(* CODESYS project projects

Project tree, tasks and I/O mapping:
  Device : CODESYS Control for Raspberry Pi SL, CODESYS GmbH, order no. 2302000009, version 4.7.0.0
    application Application
      libraries: Standard, 3.5.18.0 (System); CmpBitmapPool, * (System)
      task AC_RMP_Task (cyclic, interval t#20ms, priority 30) calls AC_PRG_RMP
      task EtherCAT_Task (cyclic, interval t#4ms, priority 1) calls nothing
      task HIGH (cyclic, interval t#5ms, priority 1) calls AC_CALL_HIGH_START, AC_CALL_HIGH_END
      task LOW (cyclic, interval t#20ms, priority 10) calls AC_CALL_LOW_START, AC_CALL_LOW_END
      task MainTask (cyclic, interval t#4ms, priority 1) calls Climate, Environment
      task TrendRecordingTask (cyclic, interval 100 ms, priority 31) calls VisuTrendStorageAccess.GlobalInstances.g_TrendRecordingManager.CyclicCall
      task VISU_TASK (cyclic, interval 100 ms, priority 31) calls VisuElems.Visu_Prg
      AC_FBs/
        function block AC_PersistenceManager [ST]
        function block AC_PersistenceManager_PersistenceChannel [ST]
      AC_RMP/
        program AC_PRG_RMP [ST]
        global variables AC_RMP
      AC_Std/
        program AC_CALL_HIGH_END [ST]
        program AC_CALL_HIGH_START [ST]
        program AC_CALL_LOW_END [ST]
        program AC_CALL_LOW_START [ST]
        function AC_Init [ST]
        function AC_InitInternal [ST]
        function AC_OnlineChange [ST]
        global variables GVL_MODULE_TREE
        global variables GVL_PersistenceManager
        global variables MODULE_INFOS
      program Climate [CFC]
      Enumerated Types/
        data type etAlarmTypes
      program Environment [CFC]
      Function Blocks/
        function block FB_Meter [ST]: rCalcAverage, rCalcMaximum, rCalcMinimum, rScaleOutput, xAlarms, xReset
      Images/
        image pool ImagePool
      Interfaces/
        interface itfMeter: rCalcAverage, rCalcMaximum, rCalcMinimum, rScaleOutput, xAlarms, xReset
      program Irrigation [CFC]
      program Lighting [CFC]
      text PersistenceConfig
      visualisation SimpleMeter
      Structured Types/
        data type stAlarm
      Trend Recording Manager
        Visualization_Trend1
      visualisation vbMeter
      program Ventilation [CFC]
      visualisation Visualization
    Camera device
      <Empty>
    EtherCAT_Master : EtherCAT Master, 3S - Smart Software Solutions GmbH, version 4.5.0.0
        settings: NetworkName = 'eth0'; NetworkName = "eth0"; SrcAddress1 = 56486; SrcAddress2 = 850751358
      EK1100 : EK1100 EtherCAT Coupler (2A E-Bus), Beckhoff Automation GmbH & Co. KG, order no. EK1100, version Revision=16#00120000
          settings: StationAlias = 0; DC sync0 cycletime = 4000; DC sync1 cycletime = 4000
        EL1018 : EL1018 8Ch. Dig. Input 24V, 10µs, Beckhoff Automation GmbH & Co. KG, order no. EL1018, version Revision=16#00120000
            settings: StationAlias = 0; DC sync0 cycletime = 4000; DC sync1 cycletime = 4000
            unmapped channels: Input, Input, Input, Input, Input, Input, Input, Input
        EL2008 : EL2008 8Ch. Dig. Output 24V, 0.5A, Beckhoff Automation GmbH & Co. KG, order no. EL2008, version Revision=16#00100000
            settings: StationAlias = 0; DC sync0 cycletime = 4000; DC sync1 cycletime = 4000
            unmapped channels: Output, Output, Output, Output, Output, Output, Output, Output
        EL3152 : EL3152 2Ch. Ana. Input 4-20mA, Beckhoff Automation GmbH & Co. KG, order no. EL3152, version Revision=16#00000000
            settings: StationAlias = 0; DC sync0 cycletime = 4000; DC sync1 cycletime = 4000
            input  Transmitter101 : INT  // Value
            unmapped channels: Status, Status, Value
    GPIOs_A_B : GPIOs A/B, 3S - Smart Software Solutions GmbH, version 4.7.0.0
        unmapped channels: digital inputs (GPIO0..GPIO31), digital outputs (GPIO0..GPIO31)
    I²C
    Onewire
      Onewire_master : Onewire master, 3S - Smart Software Solutions GmbH, version 4.7.0.0
        AmbTemp101 : DS18B20, 3S - Smart Software Solutions GmbH, version 4.7.0.0
            settings: Unique device address = '28-3ce1045748ac'
        SoilTemp101 : DS18B20, 3S - Smart Software Solutions GmbH, version 4.7.0.0
            settings: Unique device address = '28-3ce1045771af'
        SoilTemp102 : DS18B20, 3S - Smart Software Solutions GmbH, version 4.7.0.0
            settings: Unique device address = '28-3ce10457587b'
        SoilTemp103 : DS18B20, 3S - Smart Software Solutions GmbH, version 4.7.0.0
            settings: Unique device address = '28-3ce104579414'
    SoftMotion General Axis Pool
    SPI
  libraries: VisuSymbols, 4.4.0.0 (System); AC_Persistence, 4.2.0.0 (3S - Smart Software Solutions GmbH)
  5ce3da45-db07-42e7-a21c-a00fff4ed8f6|Humidity.svg
  5ce3da45-db07-42e7-a21c-a00fff4ed8f6|Humidity.svg
  5ce3da45-db07-42e7-a21c-a00fff4ed8f6|Moisture.svg
  5ce3da45-db07-42e7-a21c-a00fff4ed8f6|Moisture.svg
  5ce3da45-db07-42e7-a21c-a00fff4ed8f6|Succulents.jpg
  5ce3da45-db07-42e7-a21c-a00fff4ed8f6|Succulents.jpg
  5ce3da45-db07-42e7-a21c-a00fff4ed8f6|Thermometer.svg
  5ce3da45-db07-42e7-a21c-a00fff4ed8f6|Thermometer.svg
  AC_GENERATOR_DATA
  text list GlobalTextList
  PersistenceManager
    Channels (pChannels)
      PersistenceChannel
        ASCIIFileStorage
        Data Storage (itfDataStorage)
  text list System
*)

// Device/Application/Enumerated Types/etAlarmTypes
{attribute 'qualified_only'}
{attribute 'strict'}
TYPE etAlarmTypes :
(
	UR := 0, // Under range alarm
	LL := 1, // Low low alarm
	L := 2, // Low Alarm
	H := 3, // High Alarm
	HH := 4, // High High Alarm
	OVR := 5 // Overage Range Alarm
);
END_TYPE

// Device/Application/Structured Types/stAlarm
TYPE stAlarm :
STRUCT
	
END_STRUCT
END_TYPE

// Device/Application/AC_RMP/AC_RMP
//Code generated by Application Composer.
//Modifying generated code is not recommended!
{attribute 'global_init_slot' := '60000'}
{attribute 'init_on_onlchange'}

VAR_GLOBAL
	{attribute 'init_on_onlchange'}
	AC_RMP_Service: AC_PERSIST.AC.RMPService := (uiLocalAppID:=9744, uiNumberOfConnections:=0, pSendConnection:=0, pReceiveConnection:=0, pRMPComFB:=0);
END_VAR

// Device/Application/AC_Std/GVL_MODULE_TREE
//Code generated by Application Composer.
//Modifying generated code is not recommended!

VAR_GLOBAL
	Module_Tree: AC_PERSIST.AC.ModuleTree;
	aNodes: ARRAY[0..3] OF AC_PERSIST.AC.MNode;
	AC_Environment: AC_PERSIST.AC.MEnv;
END_VAR

// Device/Application/AC_Std/GVL_PersistenceManager
//Code generated by Application Composer.
//Modifying generated code is not recommended!
{attribute 'analysis' := '-103'}

VAR_GLOBAL
	PersistenceManager: AC_PersistenceManager;
END_VAR

// Device/Application/AC_Std/MODULE_INFOS
//Code generated by Application Composer.
//Modifying generated code is not recommended!
{attribute 'global_init_slot' := '40000'}
{attribute 'init_on_onlchange'}

VAR_GLOBAL
	{attribute 'init_on_onlchange'}
	AC_PERSIST_PersistenceManager_INFO: AC_PERSIST.AC.ModuleInfo := (pbyModuleType := ADR('AC_PERSIST.PersistenceManager'));
	{attribute 'init_on_onlchange'}
	AC_PERSIST_PersistenceChannel_INFO: AC_PERSIST.AC.ModuleInfo := (pbyModuleType := ADR('AC_PERSIST.PersistenceChannel'));
	{attribute 'init_on_onlchange'}
	AC_PERSIST_ASCIIFileStorage_INFO: AC_PERSIST.AC.ModuleInfo := (pbyModuleType := ADR('AC_PERSIST.ASCIIFileStorage'));
END_VAR

// Device/Application/AC_RMP/AC_PRG_RMP
//Code generated by Application Composer.
//Modifying generated code is not recommended!
{attribute 'analysis' := '-9'}
PROGRAM AC_PRG_RMP
VAR
    itfRmpService2 : AC_PERSIST.AC.IRmpService2 := 0;
    xStartCyclicAction : BOOL;
    xIsActionOngoing : BOOL;
    xValid : BOOL;
    xValidEnd : BOOL := TRUE;
END_VAR

//Code generated by Application Composer.
//Modifying generated code is not recommended!
__QUERYINTERFACE(AC_RMP_Service, itfRmpService2);
IF itfRmpService2 <> 0 AND xValidEnd THEN
    xValid := itfRmpService2.GetIsActionOngoing(xIsActionOngoing=>xIsActionOngoing);
    IF NOT xValid OR (xValid AND xIsActionOngoing) THEN
        xStartCyclicAction := FALSE;
    ELSE
        xStartCyclicAction := itfRmpService2.SetIsActionOngoing(TRUE);
    END_IF
ELSE
    xStartCyclicAction := TRUE;
END_IF
IF xStartCyclicAction THEN
    AC_RMP_Service.CyclicCall() ;
END_IF
IF itfRmpService2 <> 0 AND (xStartCyclicAction OR NOT xValidEnd) THEN
    xValidEnd := itfRmpService2.SetIsActionOngoing(FALSE);
END_IF

END_PROGRAM

// Device/Application/AC_Std/AC_CALL_HIGH_START
//Code generated by Application Composer.
//Modifying generated code is not recommended!
{attribute 'analysis' := '-6, -9'}
PROGRAM AC_CALL_HIGH_START

//Code generated by Application Composer.
//Modifying generated code is not recommended!
PersistenceManager.CallPrioHighStart() ;

END_PROGRAM

// Device/Application/AC_Std/AC_CALL_HIGH_END
//Code generated by Application Composer.
//Modifying generated code is not recommended!
{attribute 'analysis' := '-6, -9'}
PROGRAM AC_CALL_HIGH_END

//Code generated by Application Composer.
//Modifying generated code is not recommended!
PersistenceManager.CallPrioHighEnd() ;

END_PROGRAM

// Device/Application/AC_Std/AC_CALL_LOW_START
//Code generated by Application Composer.
//Modifying generated code is not recommended!
{attribute 'analysis' := '-6, -9'}
PROGRAM AC_CALL_LOW_START

//Code generated by Application Composer.
//Modifying generated code is not recommended!
PersistenceManager.CallPrioLowStart() ;

END_PROGRAM

// Device/Application/AC_Std/AC_CALL_LOW_END
//Code generated by Application Composer.
//Modifying generated code is not recommended!
{attribute 'analysis' := '-6, -9'}
PROGRAM AC_CALL_LOW_END

//Code generated by Application Composer.
//Modifying generated code is not recommended!
PersistenceManager.CallPrioLowEnd() ;

END_PROGRAM

// Device/Application/Climate
PROGRAM Climate
VAR
	rAmbTempSensor : ARRAY[101..103] OF fb_meter; // Ambient temperature probes
	iAmbRosemountSensor : INT; 
END_VAR

// parameter rAmbTempSensor[102].iInterval := T#5s
// parameter rAmbTempSensor[102].rOut_100 := 257
// parameter rAmbTempSensor[102].rOut_0 := -67
// parameter rAmbTempSensor[102].rIn_100 := 125
// parameter rAmbTempSensor[102].rIn_0 := -55
// parameter rAmbTempSensor[102].sDateLastServiced := ''
// parameter rAmbTempSensor[102].sSerial := ''
// parameter rAmbTempSensor[102].sUnits := ''
// parameter rAmbTempSensor[102].sDescription := ''
// parameter rAmbTempSensor[102].sName := ''
// parameter rAmbTempSensor[102].rHHLimit := 95
// parameter rAmbTempSensor[102].rHLimit := 90
// parameter rAmbTempSensor[102].rLLimit := 48
// parameter rAmbTempSensor[102].rLLLimit := 32
// parameter rAmbTempSensor[102].rURLimit := -5
// parameter rAmbTempSensor[102].tOVRAlarm := T#5s
// parameter rAmbTempSensor[102].tHHAlarm := T#5s
// parameter rAmbTempSensor[102].tHAlarm := T#5s
// parameter rAmbTempSensor[102].tLAlarm := T#5s
// parameter rAmbTempSensor[102].tLLAlarm := T#5s
// parameter rAmbTempSensor[102].tURAlarm := T#5s
rAmbTempSensor[102](xEnable := true, rIn := Transmitter101); // FB_METER
// parameter rAmbTempSensor[101].iInterval := T#5s
// parameter rAmbTempSensor[101].rOut_100 := 257
// parameter rAmbTempSensor[101].rOut_0 := -67
// parameter rAmbTempSensor[101].rIn_100 := 125
// parameter rAmbTempSensor[101].rIn_0 := -55
// parameter rAmbTempSensor[101].sDateLastServiced := ''
// parameter rAmbTempSensor[101].sSerial := ''
// parameter rAmbTempSensor[101].sUnits := ''
// parameter rAmbTempSensor[101].sDescription := ''
// parameter rAmbTempSensor[101].sName := ''
// parameter rAmbTempSensor[101].rHHLimit := 95
// parameter rAmbTempSensor[101].rHLimit := 90
// parameter rAmbTempSensor[101].rLLimit := 48
// parameter rAmbTempSensor[101].rLLLimit := 32
// parameter rAmbTempSensor[101].rURLimit := -5
// parameter rAmbTempSensor[101].tOVRAlarm := T#5s
// parameter rAmbTempSensor[101].tHHAlarm := T#5s
// parameter rAmbTempSensor[101].tHAlarm := T#5s
// parameter rAmbTempSensor[101].tLAlarm := T#5s
// parameter rAmbTempSensor[101].tLLAlarm := T#5s
// parameter rAmbTempSensor[101].tURAlarm := T#5s
rAmbTempSensor[101](xEnable := true, rIn := AmbTemp101.rTemp); // FB_METER

END_PROGRAM

// Device/Application/Function Blocks/FB_Meter
FUNCTION_BLOCK FB_Meter IMPLEMENTS itfMeter
VAR_INPUT
	xEnable : BOOL; 
	rIn : LREAL; 
	xResetCalcs : BOOL; 
END_VAR
VAR_OUTPUT
	rOut, rMin, rMax, rAvg : REAL; 
	xInAlarm, xBusy, xDone, xError : BOOL; 
	sStatus : STRING; // Status of function block
END_VAR
VAR
	tonUr, tonLL, tonL, tonH, tonHH, tonOVR : TON; 
	{attribute 'ac_persist' := 'PersistenceChannel'}
	xURActive, xLLActive, xLActive, xHActive, xHHActive, xOVRActive : BOOL; 
	rIn_PCT : REAL; // REAL INPUT EXPRESSED AS PERCENTAGE
	i : INT; 
	{attribute 'ac_persist' := 'PersistenceChannel'}
	iExecutions : DINT; 
	iMod : INT; 
END_VAR
VAR_INPUT CONSTANT
	{attribute 'parameterCategory':='Alarming'}
	tURAlarm,tLLAlarm,tLAlarm,tHAlarm,tHHAlarm,tOVRAlarm : TIME := T#5S; // Alarm Time duration
	{attribute 'ac_persist' := 'PersistenceChannel'}
	{attribute 'parameterCategory':='Alarming'}
	rURLimit : REAL := -5.0; 
    {attribute 'ac_persist' := 'PersistenceChannel'}
	{attribute 'parameterCategory':='Alarming'}
	rLLLimit : REAL := 32.0; 
	{attribute 'ac_persist' := 'PersistenceChannel'}
	{attribute 'parameterCategory':='Alarming'}
	rLLimit  : REAL := 48.0; 
	{attribute 'ac_persist' := 'PersistenceChannel'}
	{attribute 'parameterCategory':='Alarming'}
	rHLimit  : REAL := 90.0; 
	{attribute 'ac_persist' := 'PersistenceChannel'}
    {attribute 'parameterCategory':='Alarming'}
	rHHLimit : REAL := 95.0; 
	{attribute 'ac_persist' := 'PersistenceChannel'}
	{attribute 'parameterCategory':='Alarming'}
	rOVRLimit : REAL := 125; // Alarm limits
	{attribute 'ac_persist' := 'PersistenceChannel'}
	{attribute 'parameterCategory':='Alarming'}
	xarEnableAlarms: ARRAY [0..5] OF BOOL := [2(FALSE), 2(TRUE), 2(FALSE)];
	{attribute 'ac_persist' := 'PersistenceChannel'}
	{attribute 'parameterCategory':='Information'}
	sName, sDescription, sUnits, sSerial, sDateLastServiced : STRING; 
	{attribute 'ac_persist' := 'PersistenceChannel'}
	{attribute 'parameterCategory':='Scaling'}
	rIn_0 : REAL := 4; // VALUE AT 0 PERCENT INPUT
	{attribute 'ac_persist' := 'PersistenceChannel'}
	{attribute 'parameterCategory':='Scaling'}
	rIn_100 : REAL := 20; // VALUE AT 100 PERCENT INPUT
	{attribute 'ac_persist' := 'PersistenceChannel'}
	{attribute 'parameterCategory':='Scaling'}
	rOut_0 : REAL := 0; // Output at 0 percent
	{attribute 'ac_persist' := 'PersistenceChannel'}
	{attribute 'parameterCategory':='Scaling'}
	rOut_100 : REAL := 100;  // Output at 100 percent
	{attribute 'ac_persist' := 'PersistenceChannel'}
	{attribute 'parameterCategory':='Time'}
	iInterval : TIME := t#5s; 
END_VAR

// Run the calculations
// iMod := (to_int(time()) MOD TO_INT(iInterval)); 
IF TRUE (*(TO_INT(TIME()) MOD TO_INT(iInterval)) = 0*) THEN
	iExecutions := iExecutions+1; 
	rCalcAverage(rIn:=rOut,iExecutions:=iExecutions); 
	rCalcMaximum(rIn:=rOut); 
	rCalcMinimum(rin:=rOut); 
	rScaleOutput(rIn:=rIn); 
// From the list of enabled alarms, calculate the alarm expression
	FOR i:=0 TO 5 DO
		IF i<=2 THEN 
			xAlarms(rIn:=rIn,iAlarmType:=etAlarmTypes.L); 
		ELSIF i>=3 AND i<6 THEN 
			xAlarms(rIN:=rIn,iAlarmType:=etAlarmTypes.H); 
		ELSE
			; 
		END_IF	
	END_FOR
END_IF
	
IF xResetCalcs THEN 
	xReset(); 
END_IF

{warning 'Add method implementation '}
METHOD rCalcAverage : REAL
VAR_INPUT
	rIn	: REAL;
	iExecutions : DINT; 
END_VAR
VAR_OUTPUT
END_VAR
rAvg:=(rAvg*iExecutions+MAX(RAvg,rIn))/(iExecutions+1); // calculate the average of the output
END_METHOD

{warning 'Add method implementation '}
METHOD rCalcMaximum : REAL
VAR_INPUT
	rIn	: REAL;
END_VAR
IF rIn > rMax THEN 
	rMax := rIN;
ELSE 
	rMax := rMax; 
END_IF
END_METHOD

{warning 'Add method implementation '}
METHOD rCalcMinimum : REAL
VAR_INPUT
	rIn	: REAL;
END_VAR
IF rIn < rMin THEN 
	rMin := rIn; 
ELSE
	rMin := rMin; 
END_IF
END_METHOD

{warning 'Add method implementation '}
METHOD rScaleOutput : REAL
VAR_INPUT
	rIn	: REAL;
END_VAR
THIS^.rIn_PCT:=(rIn-rIn_0)/(rIn_100-rIn_0)*100; // Calculate output in percentage
this^.rOut:=THIS^.rIn_PCT/100 * (THIS^.rOut_100 - THIS^.rOut_0) + THIS^.rOut_0; // Linear scaling of output within scaling parameters
END_METHOD

{warning 'Add method implementation '}
METHOD xAlarms : BOOL
VAR_INPUT
	rIn	: REAL;
	(* Alarm Type *)
	iAlarmType	: etAlarmTypes;
END_VAR
IF iAlarmType = etAlarmTypes.L THEN 
	IF rIn <= rURLimit THEN 
		xURActive := TRUE; 
		tonUR(in:=TRUE,PT:=tURAlarm); 
	ELSIF rIn<=rLLLimit THEN 
		xLLActive := TRUE; 
		tonLL(in:=TRUE,PT:=tLLAlarm); 
	ELSIF rIn<=rLLimit THEN 
		xLActive := TRUE; 
		tonL(in:=TRUE,pt:=TLAlarm); 
	ELSE
		xURActive:=xLLActive:=xLActive:=FALSE;
		tonUR(in:=FALSE); 
	 	tonLL(in:=FALSE); 
		tonL(in:=FALSE); 
	END_IF
ELSIF iAlarmType = etAlarmTypes.H THEN 
	IF rIn >= rHLimit THEN 
		xHActive := TRUE; 
		tonH(in:=TRUE,pt:=tHAlarm); 
	ELSIF rIn >= rHHLimit THEN 
		xHHActive := TRUE; 
		tonHH(in:=TRUE,PT:=tHHAlarm); 
	ELSIF rIn >= rOVRLimit THEN 
		xOvrActive := TRUE; 
		tonOvr(in:=TRUE,PT:=tOvrAlarm); 
	ELSE
		xHActive:=xHHActive:=xOVRActive:=FALSE; 
		tonH(in:=FALSE); 
		tonHH(in:=FALSE); 
		tonOVR(in:=FALSE); 
	END_IF
END_IF
END_METHOD

{warning 'Add method implementation '}
METHOD xReset : BOOL
THIS^.iExecutions:=0; 
rOut:=rMin:=rMax:=rAvg:=0; 
xResetCalcs:=FALSE;
END_METHOD

END_FUNCTION_BLOCK

// Device/Application/Interfaces/itfMeter
INTERFACE itfMeter

METHOD rCalcAverage : REAL
VAR_INPUT
	rIn : REAL; 
	iExecutions : DINT; 
END_VAR
VAR_OUTPUT
END_VAR
END_METHOD

METHOD rCalcMaximum : REAL
VAR_INPUT
	rIn : REAL; 
END_VAR
END_METHOD

METHOD rCalcMinimum : REAL
VAR_INPUT
	rIn : REAL; 
END_VAR
END_METHOD

METHOD rScaleOutput : REAL
VAR_INPUT
	rIn : REAL; 
END_VAR
END_METHOD

METHOD xAlarms : BOOL
VAR_INPUT
	rIn : REAL; 
	iAlarmType : etAlarmTypes; // Alarm Type 
END_VAR
END_METHOD

METHOD xReset : BOOL
VAR_INPUT
END_VAR
END_METHOD

END_INTERFACE

// Device/Application/Environment
PROGRAM Environment
VAR
	xReset : BOOL; // Reset the calculations
	rSoilTempSensor : ARRAY[101..103] OF FB_Meter; // Soil temperature DS1801 probes
	rSoilTempAvg : FB_Meter; 
END_VAR

// parameter rSoilTempSensor[101].iInterval := T#5s
// parameter rSoilTempSensor[101].rOut_100 := 257
// parameter rSoilTempSensor[101].rOut_0 := -67
// parameter rSoilTempSensor[101].rIn_100 := 125
// parameter rSoilTempSensor[101].rIn_0 := -55
// parameter rSoilTempSensor[101].sDateLastServiced := ''
// parameter rSoilTempSensor[101].sSerial := ''
// parameter rSoilTempSensor[101].sUnits := ''
// parameter rSoilTempSensor[101].sDescription := ''
// parameter rSoilTempSensor[101].sName := ''
// parameter rSoilTempSensor[101].rHHLimit := 95
// parameter rSoilTempSensor[101].rHLimit := 90
// parameter rSoilTempSensor[101].rLLimit := 48
// parameter rSoilTempSensor[101].rLLLimit := 32
// parameter rSoilTempSensor[101].rURLimit := -5
// parameter rSoilTempSensor[101].tOVRAlarm := T#5s
// parameter rSoilTempSensor[101].tHHAlarm := T#5s
// parameter rSoilTempSensor[101].tHAlarm := T#5s
// parameter rSoilTempSensor[101].tLAlarm := T#5s
// parameter rSoilTempSensor[101].tLLAlarm := T#5s
// parameter rSoilTempSensor[101].tURAlarm := T#5s
rSoilTempSensor[101](xEnable := true, rIn := SoilTemp101.rTemp, xResetCalcs := xReset); // FB_METER
// parameter rSoilTempSensor[103].iInterval := T#5s
// parameter rSoilTempSensor[103].rOut_100 := 257
// parameter rSoilTempSensor[103].rOut_0 := -67
// parameter rSoilTempSensor[103].rIn_100 := 125
// parameter rSoilTempSensor[103].rIn_0 := -55
// parameter rSoilTempSensor[103].sDateLastServiced := ''
// parameter rSoilTempSensor[103].sSerial := ''
// parameter rSoilTempSensor[103].sUnits := ''
// parameter rSoilTempSensor[103].sDescription := ''
// parameter rSoilTempSensor[103].sName := ''
// parameter rSoilTempSensor[103].rHHLimit := 95
// parameter rSoilTempSensor[103].rHLimit := 90
// parameter rSoilTempSensor[103].rLLimit := 48
// parameter rSoilTempSensor[103].rLLLimit := 32
// parameter rSoilTempSensor[103].rURLimit := -5
// parameter rSoilTempSensor[103].tOVRAlarm := T#5s
// parameter rSoilTempSensor[103].tHHAlarm := T#5s
// parameter rSoilTempSensor[103].tHAlarm := T#5s
// parameter rSoilTempSensor[103].tLAlarm := T#5s
// parameter rSoilTempSensor[103].tLLAlarm := T#5s
// parameter rSoilTempSensor[103].tURAlarm := T#5s
rSoilTempSensor[103](xEnable := true, rIn := SoilTemp103.rTemp, xResetCalcs := xReset); // FB_METER
// parameter rSoilTempSensor[102].iInterval := T#5s
// parameter rSoilTempSensor[102].rOut_100 := 257
// parameter rSoilTempSensor[102].rOut_0 := -67
// parameter rSoilTempSensor[102].rIn_100 := 125
// parameter rSoilTempSensor[102].rIn_0 := -55
// parameter rSoilTempSensor[102].sDateLastServiced := ''
// parameter rSoilTempSensor[102].sSerial := ''
// parameter rSoilTempSensor[102].sUnits := ''
// parameter rSoilTempSensor[102].sDescription := ''
// parameter rSoilTempSensor[102].sName := ''
// parameter rSoilTempSensor[102].rHHLimit := 95
// parameter rSoilTempSensor[102].rHLimit := 90
// parameter rSoilTempSensor[102].rLLimit := 48
// parameter rSoilTempSensor[102].rLLLimit := 32
// parameter rSoilTempSensor[102].rURLimit := -5
// parameter rSoilTempSensor[102].tOVRAlarm := T#5s
// parameter rSoilTempSensor[102].tHHAlarm := T#5s
// parameter rSoilTempSensor[102].tHAlarm := T#5s
// parameter rSoilTempSensor[102].tLAlarm := T#5s
// parameter rSoilTempSensor[102].tLLAlarm := T#5s
// parameter rSoilTempSensor[102].tURAlarm := T#5s
rSoilTempSensor[102](xEnable := true, rIn := SoilTemp102.rTemp, xResetCalcs := xReset); // FB_METER
// parameter rSoilTempAvg.sDescription := 'Soil Temperature Avg.'
// parameter rSoilTempAvg.sName := 'TT-SOIL'
rSoilTempAvg(rIn := (rSoilTempSensor[101].rOut + rSoilTempSensor[102].rOut + rSoilTempSensor[103].rOut) / 3, xResetCalcs := xReset); // fb_meter
xReset := FALSE;

END_PROGRAM

// Device/Application/Irrigation
PROGRAM Irrigation
VAR
	SoilTemp : ARRAY[101..103] OF FB_METER; 
END_VAR

FB_METER();

END_PROGRAM

// Device/Application/Lighting
PROGRAM Lighting
VAR
END_VAR


END_PROGRAM

// Device/Application/Ventilation
PROGRAM Ventilation
VAR
END_VAR


END_PROGRAM

// Device/Application/AC_FBs/AC_PersistenceManager
//Code generated by Application Composer.
//Modifying generated code is not recommended!
FUNCTION_BLOCK AC_PersistenceManager EXTENDS AC_PERSIST.PersistenceManager
VAR_INPUT 
    INST_PersistenceChannel : AC_PersistenceManager_PersistenceChannel;
    AC_ARRAY_pChannels : ARRAY[0..0] OF AC_PERSIST.IPersistenceChannel;
END_VAR

//Code generated by Application Composer.
//Modifying generated code is not recommended!
SUPER^();

END_FUNCTION_BLOCK

// Device/Application/AC_FBs/AC_PersistenceManager_PersistenceChannel
//Code generated by Application Composer.
//Modifying generated code is not recommended!
FUNCTION_BLOCK AC_PersistenceManager_PersistenceChannel EXTENDS AC_PERSIST.PersistenceChannel
VAR_INPUT 
    INST_ASCIIFileStorage : AC_PERSIST.ASCIIFileStorage;
END_VAR

//Code generated by Application Composer.
//Modifying generated code is not recommended!
SUPER^();

END_FUNCTION_BLOCK

// Device/Application/AC_Std/AC_Init
//Code generated by Application Composer.
//Modifying generated code is not recommended!
{attribute 'linkalways'}
{attribute 'call_after_global_init_slot' := '1234'}
FUNCTION AC_Init

//Code generated by Application Composer.
//Modifying generated code is not recommended!
AC_InitInternal(FALSE);

END_FUNCTION

// Device/Application/AC_Std/AC_InitInternal
//Code generated by Application Composer.
//Modifying generated code is not recommended!
{attribute 'analysis' := '-19, -9'}
FUNCTION AC_InitInternal
VAR_INPUT
  bOnlineChange : BOOL ;
END_VAR
VAR
  hnd : AC_PERSIST.AC.ModuleHandle ;
END_VAR

//Code generated by Application Composer.
//Modifying generated code is not recommended!
AC_Environment.mtree := Module_Tree ;
AC_Environment.rmps := AC_RMP_Service ;
{IF defined(variable:AC_Environment.exts)}
	AC_Environment.exts := 0 ;
	AC_Environment.uiexts := 0 ;
{END_IF}
{IF defined(variable:AC_Environment.prsman)}
	AC_Environment.prsman := PersistenceManager;
{END_IF}
Module_Tree.Init(ADR(aNodes), 4);
hnd := Module_Tree.AddChild(0, PersistenceManager);
PersistenceManager.SetIdentification(ADR('PersistenceManager'), ADR(AC_PERSIST_PersistenceManager_INFO), 16#26102EB2, hnd, ADR(AC_Environment)) ;
hnd := Module_Tree.AddChild(PersistenceManager, PersistenceManager.INST_PersistenceChannel);
PersistenceManager.INST_PersistenceChannel.SetIdentification(ADR('PersistenceChannel'), ADR(AC_PERSIST_PersistenceChannel_INFO), 16#2610CCE8, hnd, ADR(AC_Environment)) ;
hnd := Module_Tree.AddChild(PersistenceManager.INST_PersistenceChannel, PersistenceManager.INST_PersistenceChannel.INST_ASCIIFileStorage);
PersistenceManager.INST_PersistenceChannel.INST_ASCIIFileStorage.SetIdentification(ADR('ASCIIFileStorage'), ADR(AC_PERSIST_ASCIIFileStorage_INFO), 16#26106797, hnd, ADR(AC_Environment)) ;
PersistenceManager.uiNumberOfChannels := 1;
PersistenceManager.AC_ARRAY_pChannels[0] := PersistenceManager.INST_PersistenceChannel;
PersistenceManager.pChannels := ADR(PersistenceManager.AC_ARRAY_pChannels);
PersistenceManager.INST_PersistenceChannel.tPeriodicSaving := t#5m;
PersistenceManager.INST_PersistenceChannel.xLogSaveTimeEnabled := TRUE;
PersistenceManager.INST_PersistenceChannel.itfDataStorage := PersistenceManager.INST_PersistenceChannel.INST_ASCIIFileStorage;
IF bOnlineChange THEN
    PersistenceManager.INST_PersistenceChannel.xSaveOnChange := FALSE;
    PersistenceManager.INST_PersistenceChannel.xReadVarsDuringInit := FALSE;
    PersistenceManager.INST_PersistenceChannel.xCompressTags := TRUE;
    PersistenceManager.INST_PersistenceChannel.xConsistentCopyInHighPrioTask := FALSE;
    PersistenceManager.INST_PersistenceChannel.xConvertVarsWithDifferentType := TRUE;
    PersistenceManager.INST_PersistenceChannel.xIntegrityCheckBeforeReading := TRUE;
    PersistenceManager.INST_PersistenceChannel.xSeparateArchivePerToplevelInstance := FALSE;
    PersistenceManager.INST_PersistenceChannel.xMakeDataCRCConsistencyCheck := FALSE;
    PersistenceManager.INST_PersistenceChannel.uiSavingRetriesIfCRCCisistencyCheckFails := 0;
    PersistenceManager.INST_PersistenceChannel.eAutomaticActionOnlineChange := AC_PERSIST.AutomaticActionOnlineChange.Save;
    PersistenceManager.INST_PersistenceChannel.eAutomaticActionPlcStop := AC_PERSIST.AutomaticActionPlcStop.Save;
    PersistenceManager.INST_PersistenceChannel.INST_ASCIIFileStorage.sArchive := '%CHANNEL_NAME%';
    PersistenceManager.INST_PersistenceChannel.INST_ASCIIFileStorage.xDoubleStorage := FALSE;
    PersistenceManager.INST_PersistenceChannel.INST_ASCIIFileStorage.udiMaximumFileSize := 0;
    PersistenceManager.INST_PersistenceChannel.INST_ASCIIFileStorage.bySeparator := 9;
END_IF
PersistenceManager.Init(bOnlineChange);

END_FUNCTION

// Device/Application/AC_Std/AC_OnlineChange
//Code generated by Application Composer.
//Modifying generated code is not recommended!
{attribute 'linkalways'}
{attribute 'call_after_online_change_slot' := '1234'}
FUNCTION AC_OnlineChange

//Code generated by Application Composer.
//Modifying generated code is not recommended!
PersistenceManager.OnBeforeOnlineChange();
AC_InitInternal(TRUE);
PersistenceManager.OnAfterOnlineChange();

END_FUNCTION

// Device/Application/SimpleMeter
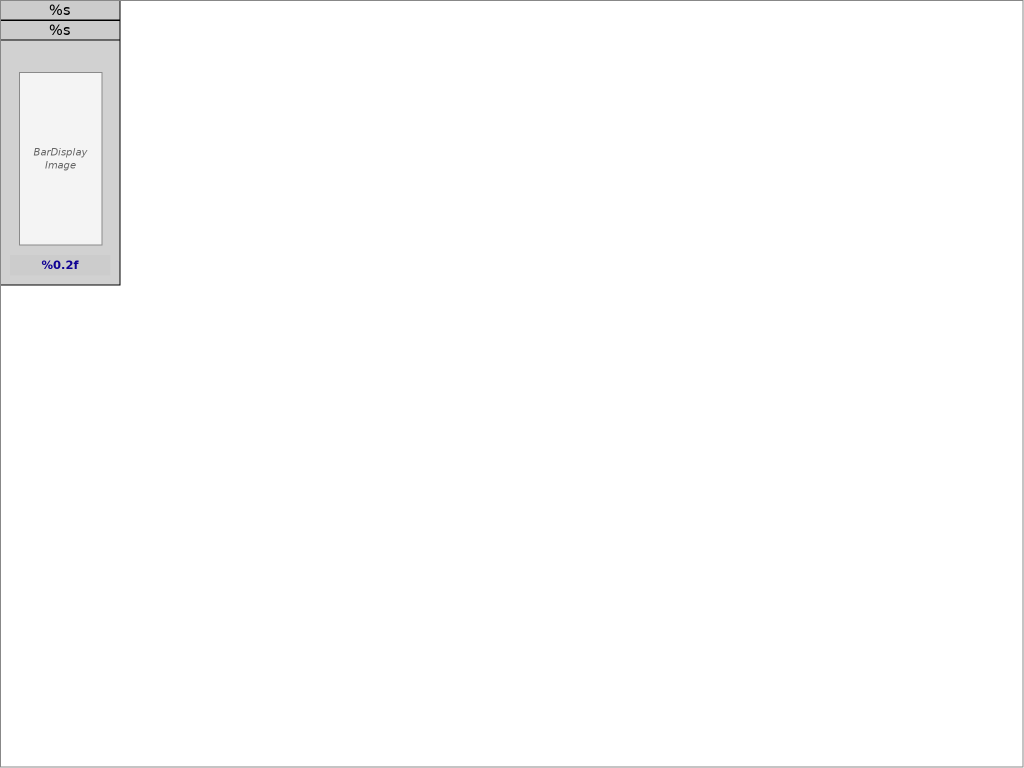
VISUALIZATION SimpleMeter  // 1024x768
VAR_IN_OUT
	meter : FB_Meter; 
END_VAR
    Rectangle (0,0 120x285), colour toggle: meter.xHActive
    BarDisplayImage (19,72 83x173), value: meter.rOut, style: BarDisplayImage-Gray, scale format: %.1f, scale 0..100
    Rectangle (0,0 120x20), "%s", text variable: meter.sName
    Rectangle (0,20 120x20), "%s", text variable: meter.sDescription
    Rectangle (10,255 100x20), "%0.2f", text variable: meter.rOut
END_VISUALIZATION

// Device/Application/vbMeter
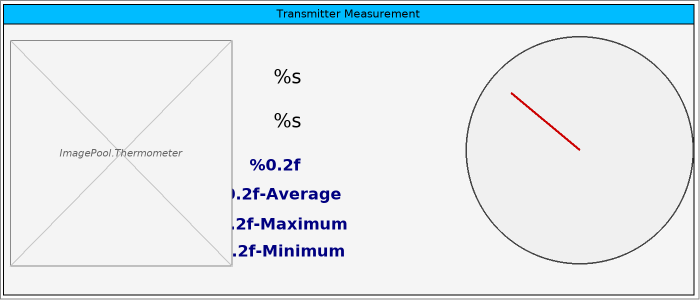
VISUALIZATION vbMeter  // 700x300
VAR_IN_OUT
	fbMeter : FB_Meter; 
END_VAR
    Rectangle (3,4 691x291)
    Rectangle (200,150 150x30), "%0.2f", text variable: fbMeter.rOut
    Rectangle (140,62 295x30), "%s", text variable: fbMeter.sName
    Rectangle (140,106 295x30), "%s", text variable: fbMeter.sDescription
    Meter360 (445,36 269x228), value: fbMeter.rOut, style: Meter-Meter360-Gray, scale format: %.1f, scale 0..100
    Rectangle (3,4 691x20), "Transmitter Measurement"
    Rectangle (200,179 150x30), "%0.2f-Average", text variable: fbMeter.rAvg
    Rectangle (200,209 150x30), "%0.2f-Maximum", text variable: fbMeter.rMax
    Rectangle (200,236 150x30), "%0.2f-Minimum", text variable: fbMeter.rMin
    Image (10,40 222x226), image: ImagePool.Thermometer
END_VISUALIZATION

// Device/Application/Visualization
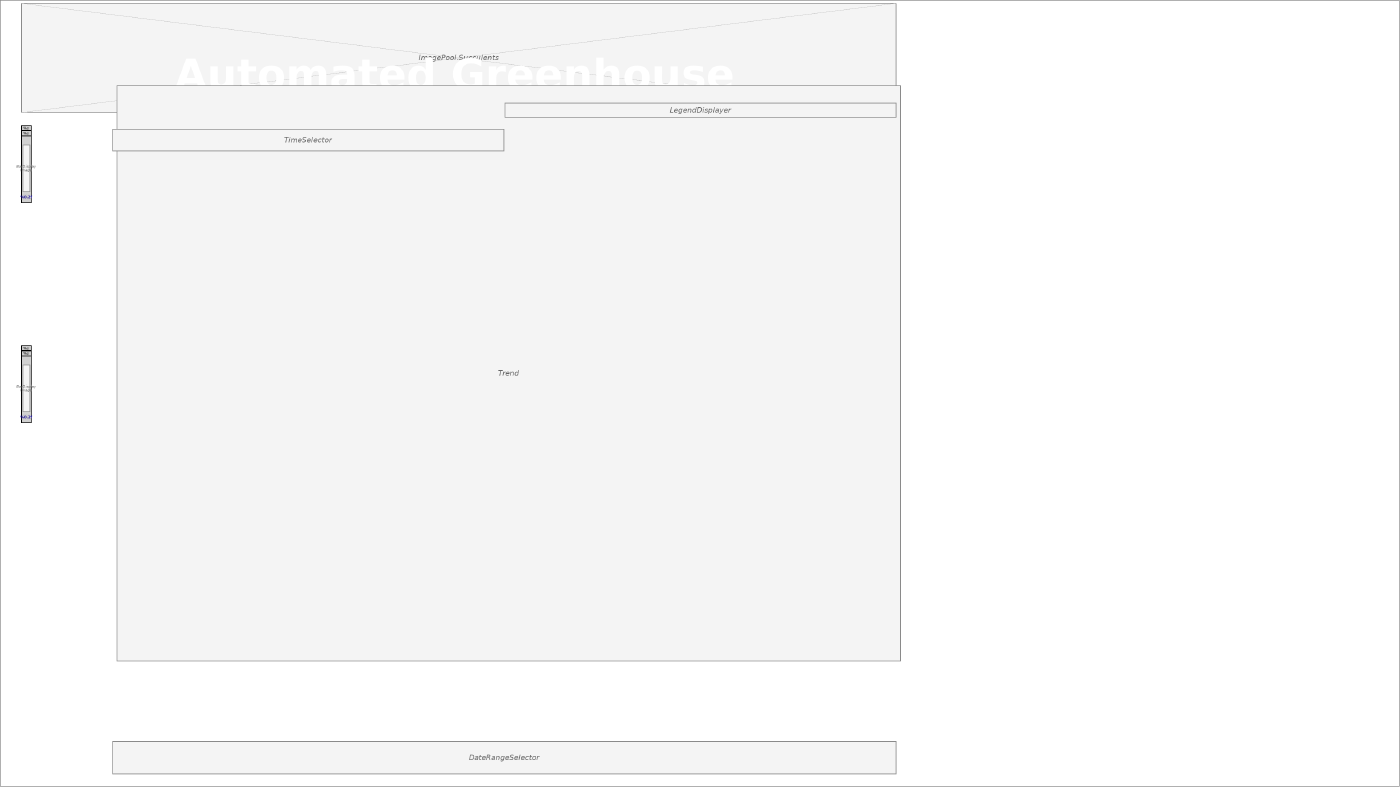
VISUALIZATION Visualization  // 1920x1080
VAR_IN_OUT
END_VAR
VAR
	bZmEnable17 : BOOL;
	bZmHome17 : BOOL;
	bZmUndo17 : BOOL;
	bIsZoomed17 : BOOL;
	bPanEnable17 : BOOL;
	bPanHome17 : BOOL;
	bIsPanned17 : BOOL;
	bEnableOnY17 : BOOL;
END_VAR
    Image (29,4 1200x150), image: ImagePool.Succulents
    Label (35,42 1177x120), "Automated Greenhouse"
    Trend (160,117 1075x790)
        p758368661: M/d/yyyy
        p2423372160: h:mm:ss tt:ms
        p2833066001: Visualization_Trend1
        p2059293862: Trend1DateRangeSelector
        p2541140726: Trend1TimeSelector
        p1690078355: Trend1Legend
        p2125894068: bZmEnable17
        p1333918548: bZmHome17
        p121640424: bZmUndo17
        p3024055206: bIsZoomed17
        p2372688541: bPanEnable17
        p4086050889: bPanHome17
        p3028486355: bIsPanned17
        p2022612088: bEnableOnY17
    Frame (29,172 121x286)
        shows SimpleMeter(meter := Climate.rAmbTempSensor[101])
    Frame (29,474 121x286)
        shows SimpleMeter(meter := Environment.rSoilTempAvg)
    DateRangeSelector (154,1017 1075x45)
        p758368661: M/d/yyyy
        p2423372160: h:mm:ss tt:ms
        p1661464551: GenElemInst_18
    TimeSelector (154,177 537x30)
        p3737533738: GenElemInst_18
        p677259794: Zoom:
    LegendDisplayer (692,141 537x20)
        p3773266362: GenElemInst_18
END_VISUALIZATION

(* text list System (id | default)
  Apr | Apr
  April | April
  Aug | Aug
  August | August
  Dec | Dec
  December | December
  Feb | Feb
  February | February
  Fri | Fri
  Friday | Friday
  Jan | Jan
  January | January
  Jul | Jul
  July | July
  Jun | Jun
  June | June
  Mar | Mar
  March | March
  May | May
  May_3Letter | May
  Mon | Mon
  Monday | Monday
  Nov | Nov
  November | November
  Oct | Oct
  October | October
  Sat | Sat
  Saturday | Saturday
  Sep | Sep
  September | September
  Sun | Sun
  Sunday | Sunday
  Thu | Thu
  Thursday | Thursday
  Tue | Tue
  Tuesday | Tuesday
  Wed | Wed
  Wednesday | Wednesday
   |  *)

(* text PersistenceConfig
// Persistence configuration for application Device.Application
// Generated automatically by GenPersistence
SEC General
  Application := Device.Application ;
  ExcludedGroups := [  ] ;
  ToplevelInstanceNames := [ PersistenceManager ] ;
  ToplevelFBPaths := [ GVL_PersistenceManager.PersistenceManager ] ;
END_SEC
SEC Channel : PersistenceChannel
  Groups := [ PersistenceChannel, Setpoints ] ;
  FBPath := PersistenceManager.INST_PersistenceChannel ;
  SeparateArchivePerToplevelInstance := False ;
  CompressTags := True ;
  MaximumFileSize := 0 ;
END_SEC
*)
